FUNCTION_BLOCK CAerationActCmd (* Basic Function Block Type *)
  (* Standard: 61499-2 *)
  (* Version 0.0, 6/10/2026, Schneider Electric, Template *)
  PACKAGE SE.Nereda;
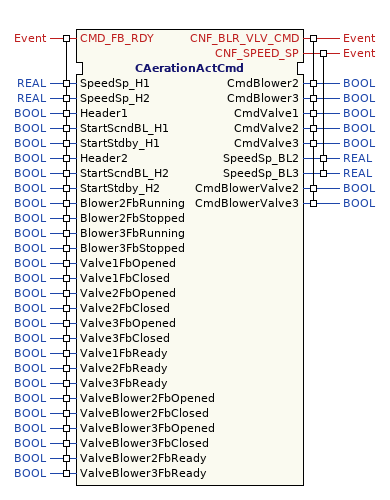
  EVENT_INPUT
    CMD_FB_RDY WITH SpeedSp_H1, SpeedSp_H2, Header1, StartScndBL_H1, StartStdby_H1, Header2, StartScndBL_H2, StartStdby_H2, Blower2FbRunning, Blower2FbStopped, Blower3FbRunning, Blower3FbStopped, Valve1FbOpened, Valve1FbClosed, Valve2FbOpened, Valve2FbClosed, Valve3FbOpened, Valve3FbClosed, Valve1FbReady, Valve2FbReady, Valve3FbReady, ValveBlower2FbOpened, ValveBlower2FbClosed, ValveBlower3FbOpened, ValveBlower3FbClosed, ValveBlower2FbReady, ValveBlower3FbReady;
  END_EVENT
  EVENT_OUTPUT
    CNF_BLR_VLV_CMD WITH CmdBlower2, CmdBlower3, CmdValve1, CmdValve2, CmdValve3, CmdBlowerValve2, CmdBlowerValve3;
    CNF_SPEED_SP WITH SpeedSp_BL2, SpeedSp_BL3;
  END_EVENT
  VAR_INPUT
    SpeedSp_H1 : REAL;
    SpeedSp_H2 : REAL;
    Header1 : BOOL;
    StartScndBL_H1 : BOOL;
    StartStdby_H1 : BOOL;
    Header2 : BOOL;
    StartScndBL_H2 : BOOL;
    StartStdby_H2 : BOOL;
    Blower2FbRunning : BOOL;
    Blower2FbStopped : BOOL;
    Blower3FbRunning : BOOL;
    Blower3FbStopped : BOOL;
    Valve1FbOpened : BOOL;
    Valve1FbClosed : BOOL;
    Valve2FbOpened : BOOL;
    Valve2FbClosed : BOOL;
    Valve3FbOpened : BOOL;
    Valve3FbClosed : BOOL;
    Valve1FbReady : BOOL;
    Valve2FbReady : BOOL;
    Valve3FbReady : BOOL;
    ValveBlower2FbOpened : BOOL;
    ValveBlower2FbClosed : BOOL;
    ValveBlower3FbOpened : BOOL;
    ValveBlower3FbClosed : BOOL;
    ValveBlower2FbReady : BOOL;
    ValveBlower3FbReady : BOOL;
  END_VAR
  VAR_OUTPUT
    CmdBlower2 : BOOL;
    CmdBlower3 : BOOL;
    CmdValve1 : BOOL;
    CmdValve2 : BOOL;
    CmdValve3 : BOOL;
    SpeedSp_BL2 : REAL;
    SpeedSp_BL3 : REAL;
    CmdBlowerValve2 : BOOL;
    CmdBlowerValve3 : BOOL;
  END_VAR
  VAR
    NormalModeR1 : BOOL;
    NormalModeR2 : BOOL;
    BlowersOk : BOOL;
  END_VAR
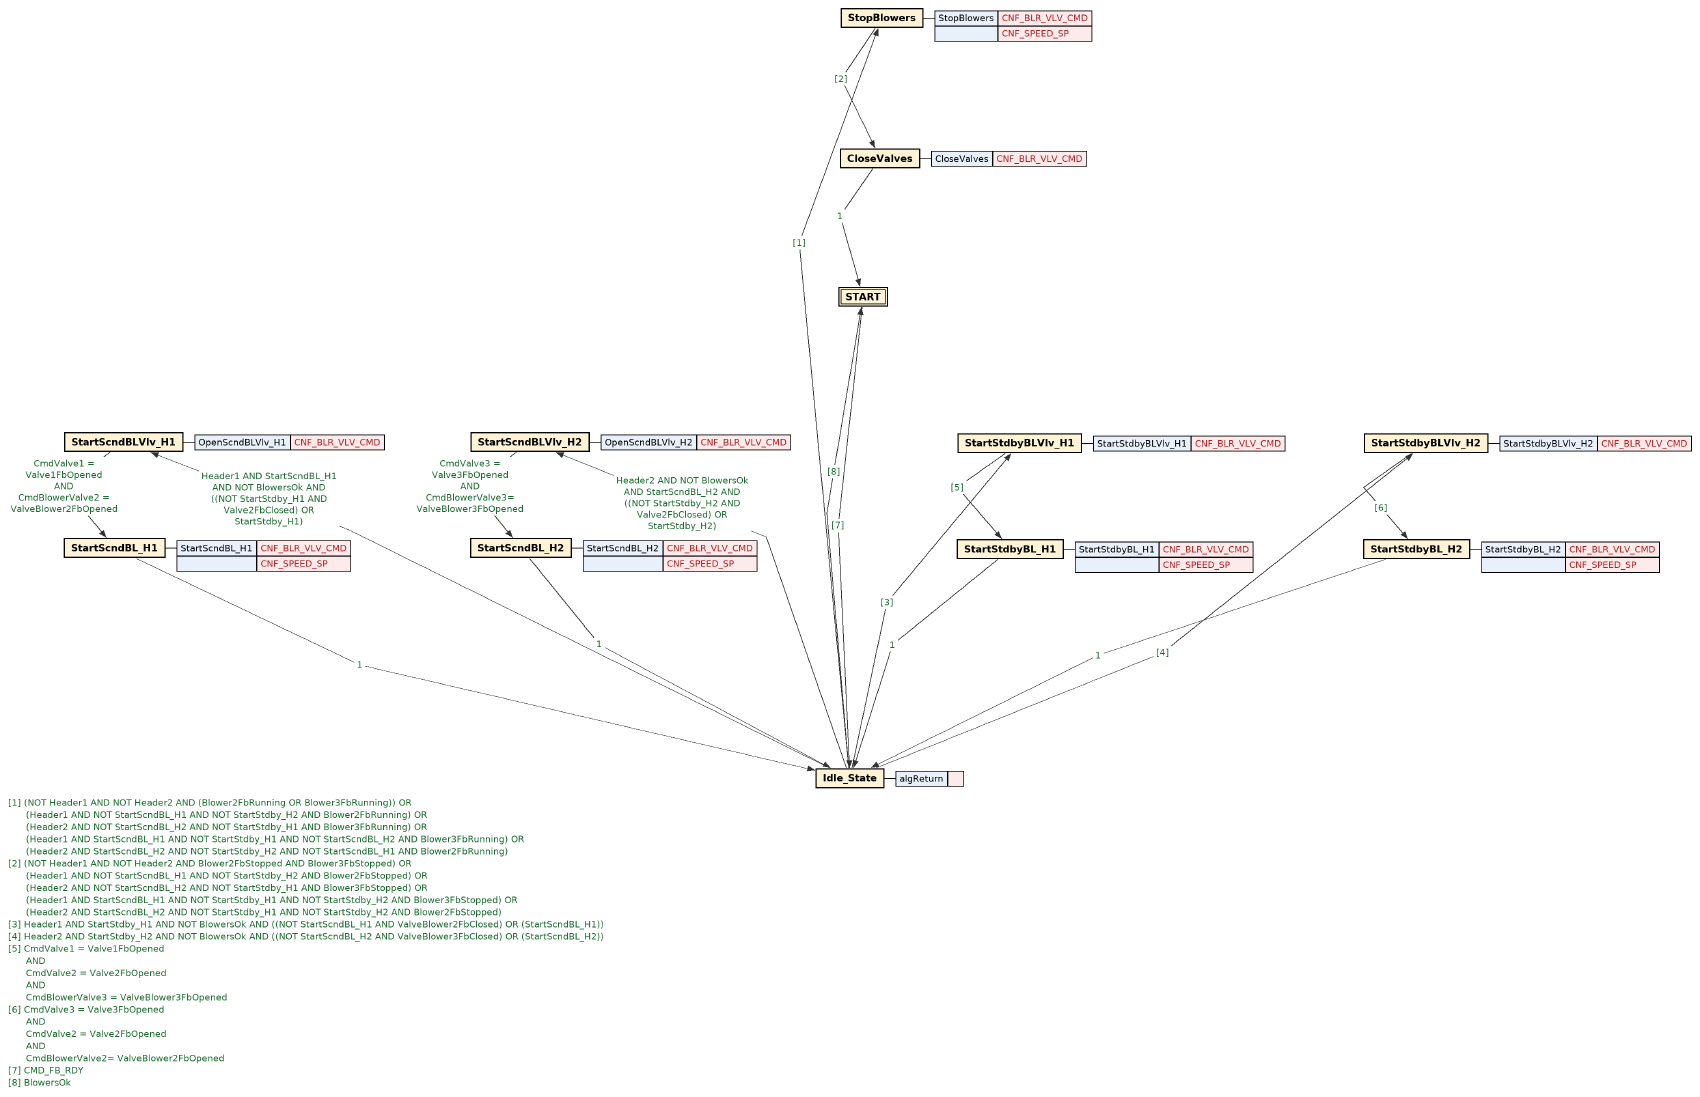
  EC_STATES
    START; (* Initial State *)
    StartScndBLVlv_H1 : OpenScndBLVlv_H1 -> CNF_BLR_VLV_CMD;
    StartScndBL_H1 : StartScndBL_H1 -> CNF_BLR_VLV_CMD, -> CNF_SPEED_SP;
    Idle_State : algReturn;
    StartScndBLVlv_H2 : OpenScndBLVlv_H2 -> CNF_BLR_VLV_CMD;
    StartScndBL_H2 : StartScndBL_H2 -> CNF_BLR_VLV_CMD, -> CNF_SPEED_SP;
    StartStdbyBLVlv_H1 : StartStdbyBLVlv_H1 -> CNF_BLR_VLV_CMD;
    StartStdbyBL_H1 : StartStdbyBL_H1 -> CNF_BLR_VLV_CMD, -> CNF_SPEED_SP;
    StartStdbyBLVlv_H2 : StartStdbyBLVlv_H2 -> CNF_BLR_VLV_CMD;
    StartStdbyBL_H2 : StartStdbyBL_H2 -> CNF_BLR_VLV_CMD, -> CNF_SPEED_SP;
    StopBlowers : StopBlowers -> CNF_BLR_VLV_CMD, -> CNF_SPEED_SP;
    CloseValves : CloseValves -> CNF_BLR_VLV_CMD;
  END_STATES
  EC_TRANSITIONS
    START TO Idle_State := CMD_FB_RDY;
    Idle_State TO StartScndBLVlv_H1 := Header1 AND StartScndBL_H1 AND NOT BlowersOk AND ((NOT StartStdby_H1 AND Valve2FbClosed) OR StartStdby_H1);
    StartScndBLVlv_H1 TO StartScndBL_H1 := CmdValve1 = Valve1FbOpened AND CmdBlowerValve2 = ValveBlower2FbOpened;
    StartScndBL_H1 TO Idle_State := 1;
    Idle_State TO StartScndBLVlv_H2 := Header2 AND NOT BlowersOk AND StartScndBL_H2 AND ((NOT StartStdby_H2 AND Valve2FbClosed) OR StartStdby_H2);
    StartScndBLVlv_H2 TO StartScndBL_H2 := CmdValve3 = Valve3FbOpened AND CmdBlowerValve3= ValveBlower3FbOpened;
    StartScndBL_H2 TO Idle_State := 1;
    Idle_State TO StartStdbyBLVlv_H1 := Header1 AND StartStdby_H1 AND NOT BlowersOk AND ((NOT StartScndBL_H1 AND ValveBlower2FbClosed) OR (StartScndBL_H1));
    StartStdbyBLVlv_H1 TO StartStdbyBL_H1 := CmdValve1 = Valve1FbOpened AND CmdValve2 = Valve2FbOpened AND CmdBlowerValve3 = ValveBlower3FbOpened;
    StartStdbyBL_H1 TO Idle_State := 1;
    Idle_State TO StartStdbyBLVlv_H2 := Header2 AND StartStdby_H2 AND NOT BlowersOk AND ((NOT StartScndBL_H2 AND ValveBlower3FbClosed) OR (StartScndBL_H2));
    StartStdbyBLVlv_H2 TO StartStdbyBL_H2 := CmdValve3 = Valve3FbOpened AND CmdValve2 = Valve2FbOpened AND CmdBlowerValve2= ValveBlower2FbOpened;
    StartStdbyBL_H2 TO Idle_State := 1;
    Idle_State TO StopBlowers := (NOT Header1 AND NOT Header2 AND (Blower2FbRunning OR Blower3FbRunning)) OR (Header1 AND NOT StartScndBL_H1 AND NOT StartStdby_H2 AND Blower2FbRunning) OR (Header2 AND NOT StartScndBL_H2 AND NOT StartStdby_H1 AND Blower3FbRunning) OR (Header1 AND StartScndBL_H1 AND NOT StartStdby_H1 AND NOT StartScndBL_H2 AND Blower3FbRunning) OR (Header2 AND StartScndBL_H2 AND NOT StartStdby_H2 AND NOT StartScndBL_H1 AND Blower2FbRunning);
    StopBlowers TO CloseValves := (NOT Header1 AND NOT Header2 AND Blower2FbStopped AND Blower3FbStopped) OR (Header1 AND NOT StartScndBL_H1 AND NOT StartStdby_H2 AND Blower2FbStopped) OR (Header2 AND NOT StartScndBL_H2 AND NOT StartStdby_H1 AND Blower3FbStopped) OR (Header1 AND StartScndBL_H1 AND NOT StartStdby_H1 AND NOT StartStdby_H2 AND Blower3FbStopped) OR (Header2 AND StartScndBL_H2 AND NOT StartStdby_H1 AND NOT StartStdby_H2 AND Blower2FbStopped);
    CloseValves TO START := 1;
    Idle_State TO START := BlowersOk;
  END_TRANSITIONS
  ALGORITHM OpenScndBLVlv_H1 IN ST:
;
CmdValve1 := TRUE;
CmdBlowerValve2 := TRUE;
  END_ALGORITHM
  ALGORITHM StartScndBL_H1 IN ST:
;
CmdBlower2 := TRUE;
SpeedSp_BL2 := SpeedSp_H1;
CMD_FB_RDY := FALSE;
  END_ALGORITHM
  ALGORITHM OpenScndBLVlv_H2 IN ST:
;
CmdValve3 := TRUE;

CmdBlowerValve3 := TRUE;
  END_ALGORITHM
  ALGORITHM StartScndBL_H2 IN ST:
;
CmdBlower3 := TRUE;
SpeedSp_BL3 := SpeedSp_H2;
CMD_FB_RDY := FALSE;
  END_ALGORITHM
  ALGORITHM StartStdbyBLVlv_H1 IN ST:
;
CmdValve1 := TRUE;
CmdValve2 := TRUE;

CmdBlowerValve3 := TRUE;
  END_ALGORITHM
  ALGORITHM StartStdbyBL_H1 IN ST:
;
CmdBlower3 := TRUE;
SpeedSp_BL3 := SpeedSp_H1;
CMD_FB_RDY := FALSE;
  END_ALGORITHM
  ALGORITHM StartStdbyBLVlv_H2 IN ST:
;
CmdValve3 := TRUE;
CmdValve2 := TRUE;

CmdBlowerValve2 := TRUE;
  END_ALGORITHM
  ALGORITHM StartStdbyBL_H2 IN ST:
;
CmdBlower2 := TRUE;
SpeedSp_BL2 := SpeedSp_H2;
CMD_FB_RDY := FALSE;
  END_ALGORITHM
  ALGORITHM StopBlowers IN ST:
;
IF NOT Header1 AND NOT Header2 THEN
	CmdBlower2 := FALSE;
	CmdBlower3 := FALSE;
END_IF;

IF Header1 AND NOT StartScndBL_H1 AND NOT StartStdby_H2 THEN
	CmdBlower2 := FALSE;
END_IF;

IF Header2 AND NOT StartScndBL_H2 AND NOT StartStdby_H1 THEN
	CmdBlower3 := FALSE;
END_IF;

IF Header1 AND StartScndBL_H1 AND NOT StartStdby_H1 AND NOT StartStdby_H2 THEN
	CmdBlower3 := FALSE;
END_IF;

IF Header2 AND StartScndBL_H2 AND NOT StartStdby_H1 AND NOT StartStdby_H2 THEN
	CmdBlower2 := FALSE;
END_IF;
  END_ALGORITHM
  ALGORITHM CloseValves IN ST:
;
IF NOT Header1 AND NOT Header2 THEN
	CmdValve1 := FALSE;
	CmdValve2 := FALSE;
	CmdValve3 := FALSE;
END_IF;

IF Header1 AND (NOT StartScndBL_H1 AND NOT StartStdby_H1) AND NOT StartStdby_H2 THEN
	CmdValve1 := FALSE;
	CmdValve2 := FALSE;
END_IF;

IF Header2 AND (NOT StartScndBL_H2 AND NOT StartStdby_H2) AND NOT StartStdby_H1 THEN
	CmdValve2 := FALSE;
	CmdValve3 := FALSE;
END_IF;

IF Header1 AND StartScndBL_H1 AND NOT StartStdby_H1 AND NOT StartStdby_H2 THEN
	CmdValve2 := FALSE;
END_IF;

IF Header2 AND StartScndBL_H2 AND NOT StartStdby_H1 AND NOT StartStdby_H2 THEN
	CmdValve2 := FALSE;
END_IF;

/*BlowerValves*/
IF NOT Header1 AND NOT Header2 THEN
	CmdBlowerValve2 := FALSE;
	CmdBlowerValve3 := FALSE;
END_IF;

IF Header1 AND NOT StartScndBL_H1 AND NOT StartStdby_H2 THEN
	CmdBlowerValve2 := FALSE;
END_IF;

IF Header2 AND NOT StartScndBL_H2 AND NOT StartStdby_H1 THEN
	CmdBlowerValve3 := FALSE;
END_IF;

IF Header1 AND StartScndBL_H1 AND NOT StartStdby_H1 AND NOT StartStdby_H2 THEN
	CmdBlowerValve3 := FALSE;
END_IF;

IF Header2 AND StartScndBL_H2 AND NOT StartStdby_H1 AND NOT StartStdby_H2 THEN
	CmdBlowerValve2 := FALSE;
END_IF;
  END_ALGORITHM
  ALGORITHM algReturn IN ST:
IF Header1 AND StartScndBL_H1 AND NOT StartStdby_H1 AND (SpeedSp_BL2 = SpeedSp_H1) THEN
	BlowersOk := CmdBlower2 AND CmdBlowerValve2 AND CmdValve1;

ELSIF Header1 AND NOT StartScndBL_H1 AND StartStdby_H1 AND (SpeedSp_BL3 = SpeedSp_H1)THEN
	BlowersOk := CmdBlower3 AND CmdBlowerValve3 AND CmdValve1 AND CmdValve2;

ELSIF Header1 AND StartScndBL_H1 AND StartStdby_H1 AND ((SpeedSp_BL2 = SpeedSp_H1) AND (SpeedSp_BL3 = SpeedSp_H1)) THEN
	BlowersOk := CmdBlower2 AND CmdBlowerValve2 AND CmdBlower3 AND
	CmdBlowerValve3 AND CmdValve1 AND CmdValve2;

ELSIF Header2 AND StartScndBL_H2 AND NOT StartStdby_H2 AND (SpeedSp_BL3 = SpeedSp_H2) THEN
	BlowersOk := CmdBlower3 AND CmdBlowerValve3 AND CmdValve3;

ELSIF Header2 AND NOT StartScndBL_H2 AND StartStdby_H2 AND (SpeedSp_BL2 = SpeedSp_H2)THEN
	BlowersOk := CmdBlower2 AND CmdBlowerValve2 AND CmdValve2 AND CmdValve3;

ELSIF Header2 AND StartScndBL_H2 AND StartStdby_H2 AND ((SpeedSp_BL2 = SpeedSp_H2) AND (SpeedSp_BL3 = SpeedSp_H2)) THEN
	BlowersOk := CmdBlower2 AND CmdBlowerValve2 AND CmdBlower3 AND
	CmdBlowerValve3 AND CmdValve2 AND CmdValve3;
ELSE
	BlowersOk := FALSE;

END_IF;
;
  END_ALGORITHM
END_FUNCTION_BLOCK
